INTERFACE I_ParameterPosition EXTENDS I_ParameterPositionGetter

{attribute 'monitoring' := 'call'}
PROPERTY Position : LREAL
SET
END_SET
END_PROPERTY

END_INTERFACE

(* stored: Version 1.1.0.1
   Itf I_ParameterPosition: Id {9a57df85-ec8d-4549-914b-3fd2a8bc008f}
   Property Position: Id {a52a54f5-e79c-49a1-b0b1-c1e423719c1b}
   Set Set: Id {31ad3580-0afa-49a0-9b06-10e9ae6327e4} *)
